FUNCTION_BLOCK TaskFB (* JADE WORKER *)
  (* Standard: 61499-1 *)
  (* Version 1.0, 2014-04-22, Ahmed, Fraunhofer IGD *)
  (* Compiler header: package fb.rt; *)
  (* Compiler Java Sun JDK 1.5.0 *)
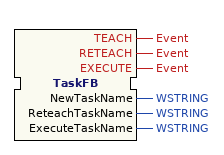
  EVENT_OUTPUT
    TEACH;
    RETEACH;
    EXECUTE;
  END_EVENT
  VAR_OUTPUT
    NewTaskName : WSTRING;
    ReteachTaskName : WSTRING;
    ExecuteTaskName : WSTRING;
  END_VAR
END_FUNCTION_BLOCK
